   1:L PR[91] R[100]mm/sec CNT100;
   1:  PR[91,1] = PR[90,1] + 31.723;
   1:  PR[91,2] = PR[90,2] + -32.039;
   1:  PR[91,3] = PR[90,3] + 104.627;
   1:L PR[91] R[100]mm/sec CNT100;
   1:  PR[91,1] = PR[90,1] + 33.260;
   1:  PR[91,2] = PR[90,2] + -32.007;
   1:  PR[91,3] = PR[90,3] + 104.643;
   1:L PR[91] R[100]mm/sec CNT100;
   1:  PR[91,1] = PR[90,1] + 37.391;
   1:  PR[91,2] = PR[90,2] + -31.583;
   1:  PR[91,3] = PR[90,3] + 104.650;
   1:L PR[91] R[100]mm/sec CNT100;
   1:  PR[91,1] = PR[90,1] + 38.518;
   1:  PR[91,2] = PR[90,2] + -31.347;
   1:  PR[91,3] = PR[90,3] + 104.671;
   1:L PR[91] R[100]mm/sec CNT100;
   1:  PR[91,1] = PR[90,1] + 42.890;
   1:  PR[91,2] = PR[90,2] + -30.128;
   1:  PR[91,3] = PR[90,3] + 104.676;
   1:L PR[91] R[100]mm/sec CNT100;
   1:  PR[91,1] = PR[90,1] + 43.497;
   1:  PR[91,2] = PR[90,2] + -29.878;
   1:  PR[91,3] = PR[90,3] + 104.698;
   1:L PR[91] R[100]mm/sec CNT100;
   1:  PR[91,1] = PR[90,1] + 48.014;
   1:  PR[91,2] = PR[90,2] + -27.738;
   1:  PR[91,3] = PR[90,3] + 104.701;
   1:L PR[91] R[100]mm/sec CNT100;
   1:  PR[91,1] = PR[90,1] + 52.491;
   1:  PR[91,2] = PR[90,2] + -24.657;
   1:  PR[91,3] = PR[90,3] + 104.726;
   1:L PR[91] R[100]mm/sec CNT100;
   1:  PR[91,1] = PR[90,1] + 52.939;
   1:  PR[91,2] = PR[90,2] + -24.278;
   1:  PR[91,3] = PR[90,3] + 104.752;
   1:L PR[91] R[100]mm/sec CNT100;
   1:  PR[91,1] = PR[90,1] + 56.290;
   1:  PR[91,2] = PR[90,2] + -21.026;
   1:  PR[91,3] = PR[90,3] + 104.755;
   1:L PR[91] R[100]mm/sec CNT100;
   1:  PR[91,1] = PR[90,1] + 57.496;
   1:  PR[91,2] = PR[90,2] + -19.555;
   1:  PR[91,3] = PR[90,3] + 104.777;
   1:L PR[91] R[100]mm/sec CNT100;
   1:  PR[91,1] = PR[90,1] + 59.518;
   1:  PR[91,2] = PR[90,2] + -16.773;
   1:  PR[91,3] = PR[90,3] + 104.787;
   1:L PR[91] R[100]mm/sec CNT100;
   1:  PR[91,1] = PR[90,1] + 61.164;
   1:  PR[91,2] = PR[90,2] + -13.760;
   1:  PR[91,3] = PR[90,3] + 104.803;
   1:L PR[91] R[100]mm/sec CNT100;
   1:  PR[91,1] = PR[90,1] + 62.061;
   1:  PR[91,2] = PR[90,2] + -11.918;
   1:  PR[91,3] = PR[90,3] + 104.820;
   1:L PR[91] R[100]mm/sec CNT100;
   1:  PR[91,1] = PR[90,1] + 63.499;
   1:  PR[91,2] = PR[90,2] + -7.353;
   1:  PR[91,3] = PR[90,3] + 104.830;
   1:L PR[91] R[100]mm/sec CNT100;
   1:  PR[91,1] = PR[90,1] + 63.732;
   1:  PR[91,2] = PR[90,2] + -6.522;
   1:  PR[91,3] = PR[90,3] + 104.853;
   1:L PR[91] R[100]mm/sec CNT100;
   1:  PR[91,1] = PR[90,1] + 63.816;
   1:  PR[91,2] = PR[90,2] + -5.600;
   1:  PR[91,3] = PR[90,3] + 104.857;
   1:L PR[91] R[100]mm/sec CNT100;
   1:  PR[91,1] = PR[90,1] + 64.322;
   1:  PR[91,2] = PR[90,2] + -0.727;
   1:  PR[91,3] = PR[90,3] + 104.862;
   1:L PR[91] R[100]mm/sec CNT100;
   1:  PR[91,1] = PR[90,1] + 63.735;
   1:  PR[91,2] = PR[90,2] + 5.053;
   1:  PR[91,3] = PR[90,3] + 104.886;
   1:L PR[91] R[100]mm/sec CNT100;
   1:  PR[91,1] = PR[90,1] + 63.499;
   1:  PR[91,2] = PR[90,2] + 5.895;
   1:  PR[91,3] = PR[90,3] + 104.914;
   1:L PR[91] R[100]mm/sec CNT100;
   1:  PR[91,1] = PR[90,1] + 62.061;
   1:  PR[91,2] = PR[90,2] + 10.459;
   1:  PR[91,3] = PR[90,3] + 104.918;
   1:L PR[91] R[100]mm/sec CNT100;
   1:  PR[91,1] = PR[90,1] + 61.163;
   1:  PR[91,2] = PR[90,2] + 12.302;
   1:  PR[91,3] = PR[90,3] + 104.941;
   1:L PR[91] R[100]mm/sec CNT100;
   1:  PR[91,1] = PR[90,1] + 59.516;
   1:  PR[91,2] = PR[90,2] + 15.317;
   1:  PR[91,3] = PR[90,3] + 104.951;
   1:L PR[91] R[100]mm/sec CNT100;
   1:  PR[91,1] = PR[90,1] + 57.492;
   1:  PR[91,2] = PR[90,2] + 18.101;
   1:  PR[91,3] = PR[90,3] + 104.968;
   1:L PR[91] R[100]mm/sec CNT100;
   1:  PR[91,1] = PR[90,1] + 56.286;
   1:  PR[91,2] = PR[90,2] + 19.572;
   1:  PR[91,3] = PR[90,3] + 104.984;
   1:L PR[91] R[100]mm/sec CNT100;
   1:  PR[91,1] = PR[90,1] + 52.930;
   1:  PR[91,2] = PR[90,2] + 22.827;
   1:  PR[91,3] = PR[90,3] + 104.994;
   1:L PR[91] R[100]mm/sec CNT100;
   1:  PR[91,1] = PR[90,1] + 52.482;
   1:  PR[91,2] = PR[90,2] + 23.205;
   1:  PR[91,3] = PR[90,3] + 105.016;
   1:L PR[91] R[100]mm/sec CNT100;
   1:  PR[91,1] = PR[90,1] + 48.001;
   1:  PR[91,2] = PR[90,2] + 26.286;
   1:  PR[91,3] = PR[90,3] + 105.019;
   1:L PR[91] R[100]mm/sec CNT100;
   1:  PR[91,1] = PR[90,1] + 43.484;
   1:  PR[91,2] = PR[90,2] + 28.423;
   1:  PR[91,3] = PR[90,3] + 105.046;
   1:L PR[91] R[100]mm/sec CNT100;
   1:  PR[91,1] = PR[90,1] + 42.877;
   1:  PR[91,2] = PR[90,2] + 28.674;
   1:  PR[91,3] = PR[90,3] + 105.070;
   1:L PR[91] R[100]mm/sec CNT100;
   1:  PR[91,1] = PR[90,1] + 38.506;
   1:  PR[91,2] = PR[90,2] + 29.891;
   1:  PR[91,3] = PR[90,3] + 105.073;
   1:L PR[91] R[100]mm/sec CNT100;
   1:  PR[91,1] = PR[90,1] + 37.377;
   1:  PR[91,2] = PR[90,2] + 30.127;
   1:  PR[91,3] = PR[90,3] + 105.095;
   1:L PR[91] R[100]mm/sec CNT100;
   1:  PR[91,1] = PR[90,1] + 33.248;
   1:  PR[91,2] = PR[90,2] + 30.548;
   1:  PR[91,3] = PR[90,3] + 105.101;
   1:L PR[91] R[100]mm/sec CNT100;
   1:  PR[91,1] = PR[90,1] + 31.709;
   1:  PR[91,2] = PR[90,2] + 30.581;
   1:  PR[91,3] = PR[90,3] + 105.121;
   1:L PR[91] R[100]mm/sec CNT100;
   1:  PR[91,1] = PR[90,1] + 27.915;
   1:  PR[91,2] = PR[90,2] + 30.327;
   1:  PR[91,3] = PR[90,3] + 105.128;
   1:L PR[91] R[100]mm/sec CNT100;
   1:  PR[91,1] = PR[90,1] + 26.644;
   1:  PR[91,2] = PR[90,2] + 30.180;
   1:  PR[91,3] = PR[90,3] + 105.147;
   1:L PR[91] R[100]mm/sec CNT100;
   1:  PR[91,1] = PR[90,1] + 26.104;
   1:  PR[91,2] = PR[90,2] + 30.092;
   1:  PR[91,3] = PR[90,3] + 105.153;
   1:L PR[91] R[100]mm/sec CNT100;
   1:  PR[91,1] = PR[90,1] + 25.544;
   1:  PR[91,2] = PR[90,2] + 30.107;
   1:  PR[91,3] = PR[90,3] + 105.155;
   1:L PR[91] R[100]mm/sec CNT100;
   1:  PR[91,1] = PR[90,1] + 24.329;
   1:  PR[91,2] = PR[90,2] + 30.087;
   1:  PR[91,3] = PR[90,3] + 105.158;
   1:L PR[91] R[100]mm/sec CNT100;
   1:  PR[91,1] = PR[90,1] + 15.055;
   1:  PR[91,2] = PR[90,2] + 29.482;
   1:  PR[91,3] = PR[90,3] + 105.164;
   1:L PR[91] R[100]mm/sec CNT100;
   1:  PR[91,1] = PR[90,1] + 14.674;
   1:  PR[91,2] = PR[90,2] + 29.410;
   1:  PR[91,3] = PR[90,3] + 105.209;
   1:L PR[91] R[100]mm/sec CNT100;
   1:  PR[91,1] = PR[90,1] + 6.614;
   1:  PR[91,2] = PR[90,2] + 28.195;
   1:  PR[91,3] = PR[90,3] + 105.211;
   1:L PR[91] R[100]mm/sec CNT100;
   1:  PR[91,1] = PR[90,1] + 2.021;
   1:  PR[91,2] = PR[90,2] + 27.161;
   1:  PR[91,3] = PR[90,3] + 105.251;
   1:L PR[91] R[100]mm/sec CNT100;
   1:  PR[91,1] = PR[90,1] + -0.771;
   1:  PR[91,2] = PR[90,2] + 26.651;
   1:  PR[91,3] = PR[90,3] + 105.273;
   1:L PR[91] R[100]mm/sec CNT100;
   1:  PR[91,1] = PR[90,1] + -9.843;
   1:  PR[91,2] = PR[90,2] + 24.252;
   1:  PR[91,3] = PR[90,3] + 105.287;
   1:L PR[91] R[100]mm/sec CNT100;
   1:  PR[91,1] = PR[90,1] + -17.871;
   1:  PR[91,2] = PR[90,2] + 21.371;
   1:  PR[91,3] = PR[90,3] + 105.333;
   1:L PR[91] R[100]mm/sec CNT100;
   1:  PR[91,1] = PR[90,1] + -24.750;
   1:  PR[91,2] = PR[90,2] + 18.099;
   1:  PR[91,3] = PR[90,3] + 105.374;
   1:L PR[91] R[100]mm/sec CNT100;
   1:  PR[91,1] = PR[90,1] + -30.389;
   1:  PR[91,2] = PR[90,2] + 14.529;
   1:  PR[91,3] = PR[90,3] + 105.411;
   1:L PR[91] R[100]mm/sec CNT100;
   1:  PR[91,1] = PR[90,1] + -34.749;
   1:  PR[91,2] = PR[90,2] + 10.761;
   1:  PR[91,3] = PR[90,3] + 105.443;
   1:L PR[91] R[100]mm/sec CNT100;
   1:  PR[91,1] = PR[90,1] + -37.797;
   1:  PR[91,2] = PR[90,2] + 6.911;
   1:  PR[91,3] = PR[90,3] + 105.471;
   1:L PR[91] R[100]mm/sec CNT100;
   1:  PR[91] = PR[90];
   1:  PR[91,1] = PR[90,1] + -37.438;
   1:  PR[91,2] = PR[90,2] + 3.095;
   1:  PR[91,3] = PR[90,3] + 106.795;
   1:L PR[91] R[100]mm/sec CNT100;
   1:  PR[91,1] = PR[90,1] + -38.021;
   1:  PR[91,2] = PR[90,2] + -0.729;
   1:  PR[91,3] = PR[90,3] + 105.516;
   1:L PR[91] R[100]mm/sec CNT100;
   1:  PR[91,1] = PR[90,1] + -37.438;
   1:  PR[91,2] = PR[90,2] + -4.554;
   1:  PR[91,3] = PR[90,3] + 105.535;
   1:L PR[91] R[100]mm/sec CNT100;
   1:  PR[91,1] = PR[90,1] + -35.649;
   1:  PR[91,2] = PR[90,2] + -8.432;
   1:  PR[91,3] = PR[90,3] + 105.554;
   1:L PR[91] R[100]mm/sec CNT100;
   1:  PR[91,1] = PR[90,1] + -32.577;
   1:  PR[91,2] = PR[90,2] + -12.315;
   1:  PR[91,3] = PR[90,3] + 105.575;
   1:L PR[91] R[100]mm/sec CNT100;
   1:  PR[91,1] = PR[90,1] + -31.486;
   1:  PR[91,2] = PR[90,2] + -13.265;
   1:  PR[91,3] = PR[90,3] + 105.599;
   1:L PR[91] R[100]mm/sec CNT100;
   1:  PR[91,1] = PR[90,1] + -28.191;
   1:  PR[91,2] = PR[90,2] + -16.108;
   1:  PR[91,3] = PR[90,3] + 105.606;
   1:L PR[91] R[100]mm/sec CNT100;
   1:  PR[91,1] = PR[90,1] + -22.512;
   1:  PR[91,2] = PR[90,2] + -19.706;
   1:  PR[91,3] = PR[90,3] + 105.628;
   1:L PR[91] R[100]mm/sec CNT100;
   1:  PR[91,1] = PR[90,1] + -15.586;
   1:  PR[91,2] = PR[90,2] + -23.002;
   1:  PR[91,3] = PR[90,3] + 105.660;
   1:L PR[91] R[100]mm/sec CNT100;
   1:  PR[91,1] = PR[90,1] + -7.503;
   1:  PR[91,2] = PR[90,2] + -25.906;
   1:  PR[91,3] = PR[90,3] + 105.698;
   1:L PR[91] R[100]mm/sec CNT100;
   1:  PR[91,1] = PR[90,1] + 1.762;
   1:  PR[91,2] = PR[90,2] + -28.366;
   1:  PR[91,3] = PR[90,3] + 105.740;
   1:L PR[91] R[100]mm/sec CNT100;
   1:  PR[91,1] = PR[90,1] + 7.941;
   1:  PR[91,2] = PR[90,2] + -29.756;
   1:  PR[91,3] = PR[90,3] + 105.787;
   1:L PR[91] R[100]mm/sec CNT100;
   1:  PR[91,1] = PR[90,1] + 13.802;
   1:  PR[91,2] = PR[90,2] + -30.639;
   1:  PR[91,3] = PR[90,3] + 105.818;
   1:L PR[91] R[100]mm/sec CNT100;
   1:  PR[91,1] = PR[90,1] + 16.569;
   1:  PR[91,2] = PR[90,2] + -31.163;
   1:  PR[91,3] = PR[90,3] + 105.847;
   1:L PR[91] R[100]mm/sec CNT100;
   1:  PR[91,1] = PR[90,1] + 25.855;
   1:  PR[91,2] = PR[90,2] + -31.775;
   1:  PR[91,3] = PR[90,3] + 105.861;
   1:L PR[91] R[100]mm/sec CNT100;
   1:  PR[91,1] = PR[90,1] + 26.725;
   1:  PR[91,2] = PR[90,2] + -31.791;
   1:  PR[91,3] = PR[90,3] + 105.907;
   1:L PR[91] R[100]mm/sec CNT100;
   1:  PR[91,1] = PR[90,1] + 27.669;
   1:  PR[91,2] = PR[90,2] + -31.899;
   1:  PR[91,3] = PR[90,3] + 105.911;
   1:L PR[91] R[100]mm/sec CNT100;
   1:  PR[91,1] = PR[90,1] + 32.407;
   1:  PR[91,2] = PR[90,2] + -32.212;
   1:  PR[91,3] = PR[90,3] + 105.916;
   1:L PR[91] R[100]mm/sec CNT100;
   1:  PR[91,1] = PR[90,1] + 32.895;
   1:  PR[91,2] = PR[90,2] + -32.202;
   1:  PR[91,3] = PR[90,3] + 105.939;
   1:L PR[91] R[100]mm/sec CNT100;
   1:  PR[91,1] = PR[90,1] + 38.092;
   1:  PR[91,2] = PR[90,2] + -31.668;
   1:  PR[91,3] = PR[90,3] + 105.941;
   1:L PR[91] R[100]mm/sec CNT100;
   1:  PR[91,1] = PR[90,1] + 43.282;
   1:  PR[91,2] = PR[90,2] + -30.250;
   1:  PR[91,3] = PR[90,3] + 105.967;
   1:L PR[91] R[100]mm/sec CNT100;
   1:  PR[91,1] = PR[90,1] + 43.736;
   1:  PR[91,2] = PR[90,2] + -30.088;
   1:  PR[91,3] = PR[90,3] + 105.993;
   1:L PR[91] R[100]mm/sec CNT100;
   1:  PR[91,1] = PR[90,1] + 48.043;
   1:  PR[91,2] = PR[90,2] + -28.096;
   1:  PR[91,3] = PR[90,3] + 105.996;
   1:L PR[91] R[100]mm/sec CNT100;
   1:  PR[91,1] = PR[90,1] + 49.407;
   1:  PR[91,2] = PR[90,2] + -27.311;
   1:  PR[91,3] = PR[90,3] + 106.019;
   1:L PR[91] R[100]mm/sec CNT100;
   1:  PR[91,1] = PR[90,1] + 52.446;
   1:  PR[91,2] = PR[90,2] + -25.229;
   1:  PR[91,3] = PR[90,3] + 106.027;
   1:L PR[91] R[100]mm/sec CNT100;
   1:  PR[91,1] = PR[90,1] + 54.789;
   1:  PR[91,2] = PR[90,2] + -23.251;
   1:  PR[91,3] = PR[90,3] + 106.045;
   1:L PR[91] R[100]mm/sec CNT100;
   1:  PR[91,1] = PR[90,1] + 56.409;
   1:  PR[91,2] = PR[90,2] + -21.678;
   1:  PR[91,3] = PR[90,3] + 106.060;
   1:L PR[91] R[100]mm/sec CNT100;
   1:  PR[91,1] = PR[90,1] + 59.575;
   1:  PR[91,2] = PR[90,2] + -17.816;
   1:  PR[91,3] = PR[90,3] + 106.071;
   1:L PR[91] R[100]mm/sec CNT100;
   1:  PR[91,1] = PR[90,1] + 59.849;
   1:  PR[91,2] = PR[90,2] + -17.438;
   1:  PR[91,3] = PR[90,3] + 106.095;
   1:L PR[91] R[100]mm/sec CNT100;
   1:  PR[91,1] = PR[90,1] + 60.871;
   1:  PR[91,2] = PR[90,2] + -15.568;
   1:  PR[91,3] = PR[90,3] + 106.098;
   1:L PR[91] R[100]mm/sec CNT100;
   1:  PR[91,1] = PR[90,1] + 62.396;
   1:  PR[91,2] = PR[90,2] + -12.864;
   1:  PR[91,3] = PR[90,3] + 106.108;
   1:L PR[91] R[100]mm/sec CNT100;
   1:  PR[91,1] = PR[90,1] + 62.780;
   1:  PR[91,2] = PR[90,2] + -12.209;
   1:  PR[91,3] = PR[90,3] + 106.123;
   1:L PR[91] R[100]mm/sec CNT100;
   1:  PR[91,1] = PR[90,1] + 63.948;
   1:  PR[91,2] = PR[90,2] + -8.607;
   1:  PR[91,3] = PR[90,3] + 106.127;
   1:L PR[91] R[100]mm/sec CNT100;
   1:  PR[91,1] = PR[90,1] + 64.641;
   1:  PR[91,2] = PR[90,2] + -6.555;
   1:  PR[91,3] = PR[90,3] + 106.146;
   1:L PR[91] R[100]mm/sec CNT100;
   1:  PR[91,1] = PR[90,1] + 65.278;
   1:  PR[91,2] = PR[90,2] + -0.729;
   1:  PR[91,3] = PR[90,3] + 106.156;
   1:L PR[91] R[100]mm/sec CNT100;
   1:  PR[91,1] = PR[90,1] + 64.641;
   1:  PR[91,2] = PR[90,2] + 5.096;
   1:  PR[91,3] = PR[90,3] + 106.185;
   1:L PR[91] R[100]mm/sec CNT100;
   1:  PR[91,1] = PR[90,1] + 63.948;
   1:  PR[91,2] = PR[90,2] + 7.149;
   1:  PR[91,3] = PR[90,3] + 106.214;
   1:L PR[91] R[100]mm/sec CNT100;
   1:  PR[91,1] = PR[90,1] + 62.780;
   1:  PR[91,2] = PR[90,2] + 10.749;
   1:  PR[91,3] = PR[90,3] + 106.224;
   1:L PR[91] R[100]mm/sec CNT100;
   1:  PR[91,1] = PR[90,1] + 62.396;
   1:  PR[91,2] = PR[90,2] + 11.404;
   1:  PR[91,3] = PR[90,3] + 106.243;
   1:L PR[91] R[100]mm/sec CNT100;
   1:  PR[91,1] = PR[90,1] + 60.871;
   1:  PR[91,2] = PR[90,2] + 14.110;
   1:  PR[91,3] = PR[90,3] + 106.247;
   1:L PR[91] R[100]mm/sec CNT100;
   1:  PR[91,1] = PR[90,1] + 59.850;
   1:  PR[91,2] = PR[90,2] + 15.978;
   1:  PR[91,3] = PR[90,3] + 106.262;
   1:L PR[91] R[100]mm/sec CNT100;
   1:  PR[91,1] = PR[90,1] + 59.576;
   1:  PR[91,2] = PR[90,2] + 16.356;
   1:  PR[91,3] = PR[90,3] + 106.272;
   1:L PR[91] R[100]mm/sec CNT100;
   1:  PR[91,1] = PR[90,1] + 56.408;
   1:  PR[91,2] = PR[90,2] + 20.220;
   1:  PR[91,3] = PR[90,3] + 106.274;
   1:L PR[91] R[100]mm/sec CNT100;
   1:  PR[91,1] = PR[90,1] + 54.786;
   1:  PR[91,2] = PR[90,2] + 21.794;
   1:  PR[91,3] = PR[90,3] + 106.299;
   1:L PR[91] R[100]mm/sec CNT100;
   1:  PR[91,1] = PR[90,1] + 52.441;
   1:  PR[91,2] = PR[90,2] + 23.774;
   1:  PR[91,3] = PR[90,3] + 106.310;
   1:L PR[91] R[100]mm/sec CNT100;
   1:  PR[91,1] = PR[90,1] + 49.399;
   1:  PR[91,2] = PR[90,2] + 25.857;
   1:  PR[91,3] = PR[90,3] + 106.325;
   1:L PR[91] R[100]mm/sec CNT100;
   1:  PR[91,1] = PR[90,1] + 48.034;
   1:  PR[91,2] = PR[90,2] + 26.643;
   1:  PR[91,3] = PR[90,3] + 106.343;
   1:L PR[91] R[100]mm/sec CNT100;
   1:  PR[91,1] = PR[90,1] + 43.721;
   1:  PR[91,2] = PR[90,2] + 28.634;
   1:  PR[91,3] = PR[90,3] + 106.351;
   1:L PR[91] R[100]mm/sec CNT100;
   1:  PR[91,1] = PR[90,1] + 43.269;
   1:  PR[91,2] = PR[90,2] + 28.796;
   1:  PR[91,3] = PR[90,3] + 106.374;
   1:L PR[91] R[100]mm/sec CNT100;
   1:  PR[91,1] = PR[90,1] + 38.028;
   1:  PR[91,2] = PR[90,2] + 30.218;
   1:  PR[91,3] = PR[90,3] + 106.377;
   1:L PR[91] R[100]mm/sec CNT100;
   1:  PR[91,1] = PR[90,1] + 32.877;
   1:  PR[91,2] = PR[90,2] + 30.743;
   1:  PR[91,3] = PR[90,3] + 106.403;
   1:L PR[91] R[100]mm/sec CNT100;
   1:  PR[91,1] = PR[90,1] + 32.386;
   1:  PR[91,2] = PR[90,2] + 30.754;
   1:  PR[91,3] = PR[90,3] + 106.429;
   1:L PR[91] R[100]mm/sec CNT100;
   1:  PR[91,1] = PR[90,1] + 27.651;
   1:  PR[91,2] = PR[90,2] + 30.438;
   1:  PR[91,3] = PR[90,3] + 106.431;
   1:L PR[91] R[100]mm/sec CNT100;
   1:  PR[91,1] = PR[90,1] + 26.723;
   1:  PR[91,2] = PR[90,2] + 30.330;
   1:  PR[91,3] = PR[90,3] + 106.454;
   1:L PR[91] R[100]mm/sec CNT100;
   1:  PR[91,1] = PR[90,1] + 25.868;
   1:  PR[91,2] = PR[90,2] + 30.317;
   1:  PR[91,3] = PR[90,3] + 106.459;
   1:L PR[91] R[100]mm/sec CNT100;
   1:  PR[91,1] = PR[90,1] + 16.575;
   1:  PR[91,2] = PR[90,2] + 29.705;
   1:  PR[91,3] = PR[90,3] + 106.463;
   1:L PR[91] R[100]mm/sec CNT100;
   1:  PR[91,1] = PR[90,1] + 13.802;
   1:  PR[91,2] = PR[90,2] + 29.181;
   1:  PR[91,3] = PR[90,3] + 106.509;
   1:L PR[91] R[100]mm/sec CNT100;
   1:  PR[91,1] = PR[90,1] + 7.941;
   1:  PR[91,2] = PR[90,2] + 28.297;
   1:  PR[91,3] = PR[90,3] + 106.523;
   1:L PR[91] R[100]mm/sec CNT100;
   1:  PR[91,1] = PR[90,1] + 1.762;
   1:  PR[91,2] = PR[90,2] + 26.907;
   1:  PR[91,3] = PR[90,3] + 106.552;
   1:L PR[91] R[100]mm/sec CNT100;
   1:  PR[91,1] = PR[90,1] + -7.503;
   1:  PR[91,2] = PR[90,2] + 24.448;
   1:  PR[91,3] = PR[90,3] + 106.583;
   1:L PR[91] R[100]mm/sec CNT100;
   1:  PR[91,1] = PR[90,1] + -15.586;
   1:  PR[91,2] = PR[90,2] + 21.544;
   1:  PR[91,3] = PR[90,3] + 106.630;
   1:L PR[91] R[100]mm/sec CNT100;
   1:  PR[91,1] = PR[90,1] + -22.512;
   1:  PR[91,2] = PR[90,2] + 18.247;
   1:  PR[91,3] = PR[90,3] + 106.672;
   1:L PR[91] R[100]mm/sec CNT100;
   1:  PR[91,1] = PR[90,1] + -28.190;
   1:  PR[91,2] = PR[90,2] + 14.650;
   1:  PR[91,3] = PR[90,3] + 106.709;
   1:L PR[91] R[100]mm/sec CNT100;
   1:  PR[91,1] = PR[90,1] + -32.579;
   1:  PR[91,2] = PR[90,2] + 10.853;
   1:  PR[91,3] = PR[90,3] + 106.742;
   1:L PR[91] R[100]mm/sec CNT100;
   1:  PR[91,1] = PR[90,1] + -35.649;
   1:  PR[91,2] = PR[90,2] + 6.973;
   1:  PR[91,3] = PR[90,3] + 106.771;
   1:L PR[91] R[100]mm/sec CNT100;
   1:  PR[91] = PR[90];
   1:  PR[91,1] = PR[90,1] + -35.303;
   1:  PR[91,2] = PR[90,2] + 3.126;
   1:  PR[91,3] = PR[90,3] + 108.095;
   1:L PR[91] R[100]mm/sec CNT100;
   1:  PR[91,1] = PR[90,1] + -35.891;
   1:  PR[91,2] = PR[90,2] + -0.729;
   1:  PR[91,3] = PR[90,3] + 106.816;
   1:L PR[91] R[100]mm/sec CNT100;
   1:  PR[91,1] = PR[90,1] + -35.303;
   1:  PR[91,2] = PR[90,2] + -4.585;
   1:  PR[91,3] = PR[90,3] + 106.836;
   1:L PR[91] R[100]mm/sec CNT100;
   1:  PR[91,1] = PR[90,1] + -33.501;
   1:  PR[91,2] = PR[90,2] + -8.494;
   1:  PR[91,3] = PR[90,3] + 106.855;
   1:L PR[91] R[100]mm/sec CNT100;
   1:  PR[91,1] = PR[90,1] + -30.408;
   1:  PR[91,2] = PR[90,2] + -12.406;
   1:  PR[91,3] = PR[90,3] + 106.876;
   1:L PR[91] R[100]mm/sec CNT100;
   1:  PR[91,1] = PR[90,1] + -28.966;
   1:  PR[91,2] = PR[90,2] + -13.661;
   1:  PR[91,3] = PR[90,3] + 106.901;
   1:L PR[91] R[100]mm/sec CNT100;
   1:  PR[91,1] = PR[90,1] + -25.991;
   1:  PR[91,2] = PR[90,2] + -16.228;
   1:  PR[91,3] = PR[90,3] + 106.910;
   1:L PR[91] R[100]mm/sec CNT100;
   1:  PR[91,1] = PR[90,1] + -20.274;
   1:  PR[91,2] = PR[90,2] + -19.853;
   1:  PR[91,3] = PR[90,3] + 106.930;
   1:L PR[91] R[100]mm/sec CNT100;
   1:  PR[91,1] = PR[90,1] + -13.301;
   1:  PR[91,2] = PR[90,2] + -23.175;
   1:  PR[91,3] = PR[90,3] + 106.963;
   1:L PR[91] R[100]mm/sec CNT100;
   1:  PR[91,1] = PR[90,1] + -5.165;
   1:  PR[91,2] = PR[90,2] + -26.102;
   1:  PR[91,3] = PR[90,3] + 107.001;
   1:L PR[91] R[100]mm/sec CNT100;
   1:  PR[91,1] = PR[90,1] + 0.887;
   1:  PR[91,2] = PR[90,2] + -27.704;
   1:  PR[91,3] = PR[90,3] + 107.044;
   1:L PR[91] R[100]mm/sec CNT100;
   1:  PR[91,1] = PR[90,1] + 2.723;
   1:  PR[91,2] = PR[90,2] + -28.294;
   1:  PR[91,3] = PR[90,3] + 107.075;
   1:L PR[91] R[100]mm/sec CNT100;
   1:  PR[91,1] = PR[90,1] + 5.426;
   1:  PR[91,2] = PR[90,2] + -28.994;
   1:  PR[91,3] = PR[90,3] + 107.085;
   1:L PR[91] R[100]mm/sec CNT100;
   1:  PR[91,1] = PR[90,1] + 9.267;
   1:  PR[91,2] = PR[90,2] + -29.858;
   1:  PR[91,3] = PR[90,3] + 107.098;
   1:L PR[91] R[100]mm/sec CNT100;
   1:  PR[91,1] = PR[90,1] + 12.931;
   1:  PR[91,2] = PR[90,2] + -30.410;
   1:  PR[91,3] = PR[90,3] + 107.118;
   1:L PR[91] R[100]mm/sec CNT100;
   1:  PR[91,1] = PR[90,1] + 18.085;
   1:  PR[91,2] = PR[90,2] + -31.386;
   1:  PR[91,3] = PR[90,3] + 107.136;
   1:L PR[91] R[100]mm/sec CNT100;
   1:  PR[91,1] = PR[90,1] + 32.755;
   1:  PR[91,2] = PR[90,2] + -32.361;
   1:  PR[91,3] = PR[90,3] + 107.162;
   1:L PR[91] R[100]mm/sec CNT100;
   1:  PR[91,1] = PR[90,1] + 33.002;
   1:  PR[91,2] = PR[90,2] + -32.363;
   1:  PR[91,3] = PR[90,3] + 107.235;
   1:L PR[91] R[100]mm/sec CNT100;
   1:  PR[91,1] = PR[90,1] + 37.963;
   1:  PR[91,2] = PR[90,2] + -31.870;
   1:  PR[91,3] = PR[90,3] + 107.236;
   1:L PR[91] R[100]mm/sec CNT100;
   1:  PR[91,1] = PR[90,1] + 38.977;
   1:  PR[91,2] = PR[90,2] + -31.699;
   1:  PR[91,3] = PR[90,3] + 107.261;
   1:L PR[91] R[100]mm/sec CNT100;
   1:  PR[91,1] = PR[90,1] + 43.040;
   1:  PR[91,2] = PR[90,2] + -30.595;
   1:  PR[91,3] = PR[90,3] + 107.266;
   1:L PR[91] R[100]mm/sec CNT100;
   1:  PR[91,1] = PR[90,1] + 45.009;
   1:  PR[91,2] = PR[90,2] + -29.889;
   1:  PR[91,3] = PR[90,3] + 107.287;
   1:L PR[91] R[100]mm/sec CNT100;
   1:  PR[91,1] = PR[90,1] + 47.878;
   1:  PR[91,2] = PR[90,2] + -28.562;
   1:  PR[91,3] = PR[90,3] + 107.297;
   1:L PR[91] R[100]mm/sec CNT100;
   1:  PR[91,1] = PR[90,1] + 50.965;
   1:  PR[91,2] = PR[90,2] + -26.786;
   1:  PR[91,3] = PR[90,3] + 107.313;
   1:L PR[91] R[100]mm/sec CNT100;
   1:  PR[91,1] = PR[90,1] + 52.399;
   1:  PR[91,2] = PR[90,2] + -25.803;
   1:  PR[91,3] = PR[90,3] + 107.330;
   1:L PR[91] R[100]mm/sec CNT100;
   1:  PR[91,1] = PR[90,1] + 56.564;
   1:  PR[91,2] = PR[90,2] + -22.286;
   1:  PR[91,3] = PR[90,3] + 107.339;
   1:L PR[91] R[100]mm/sec CNT100;
   1:  PR[91,1] = PR[90,1] + 59.657;
   1:  PR[91,2] = PR[90,2] + -18.639;
   1:  PR[91,3] = PR[90,3] + 107.366;
   1:L PR[91] R[100]mm/sec CNT100;
   1:  PR[91,1] = PR[90,1] + 60.635;
   1:  PR[91,2] = PR[90,2] + -17.521;
   1:  PR[91,3] = PR[90,3] + 107.389;
   1:L PR[91] R[100]mm/sec CNT100;
   1:  PR[91,1] = PR[90,1] + 61.969;
   1:  PR[91,2] = PR[90,2] + -15.155;
   1:  PR[91,3] = PR[90,3] + 107.397;
   1:L PR[91] R[100]mm/sec CNT100;
   1:  PR[91,1] = PR[90,1] + 63.685;
   1:  PR[91,2] = PR[90,2] + -12.224;
   1:  PR[91,3] = PR[90,3] + 107.410;
   1:L PR[91] R[100]mm/sec CNT100;
   1:  PR[91,1] = PR[90,1] + 64.460;
   1:  PR[91,2] = PR[90,2] + -9.904;
   1:  PR[91,3] = PR[90,3] + 107.427;
   1:L PR[91] R[100]mm/sec CNT100;
   1:  PR[91,1] = PR[90,1] + 65.455;
   1:  PR[91,2] = PR[90,2] + -7.038;
   1:  PR[91,3] = PR[90,3] + 107.439;
   1:L PR[91] R[100]mm/sec CNT100;
   1:  PR[91,1] = PR[90,1] + 65.654;
   1:  PR[91,2] = PR[90,2] + -6.234;
   1:  PR[91,3] = PR[90,3] + 107.454;
   1:L PR[91] R[100]mm/sec CNT100;
   1:  PR[91,1] = PR[90,1] + 66.079;
   1:  PR[91,2] = PR[90,2] + -2.515;
   1:  PR[91,3] = PR[90,3] + 107.458;
   1:L PR[91] R[100]mm/sec CNT100;
   1:  PR[91,1] = PR[90,1] + 66.226;
   1:  PR[91,2] = PR[90,2] + -0.755;
   1:  PR[91,3] = PR[90,3] + 107.477;
   1:L PR[91] R[100]mm/sec CNT100;
   1:  PR[91,1] = PR[90,1] + 65.763;
   1:  PR[91,2] = PR[90,2] + 3.477;
   1:  PR[91,3] = PR[90,3] + 107.485;
   1:L PR[91] R[100]mm/sec CNT100;
   1:  PR[91,1] = PR[90,1] + 65.647;
   1:  PR[91,2] = PR[90,2] + 4.802;
   1:  PR[91,3] = PR[90,3] + 107.507;
   1:L PR[91] R[100]mm/sec CNT100;
   1:  PR[91,1] = PR[90,1] + 65.455;
   1:  PR[91,2] = PR[90,2] + 5.580;
   1:  PR[91,3] = PR[90,3] + 107.513;
   1:L PR[91] R[100]mm/sec CNT100;
   1:  PR[91,1] = PR[90,1] + 64.460;
   1:  PR[91,2] = PR[90,2] + 8.445;
   1:  PR[91,3] = PR[90,3] + 107.517;
   1:L PR[91] R[100]mm/sec CNT100;
   1:  PR[91,1] = PR[90,1] + 63.684;
   1:  PR[91,2] = PR[90,2] + 10.767;
   1:  PR[91,3] = PR[90,3] + 107.532;
   1:L PR[91] R[100]mm/sec CNT100;
   1:  PR[91,1] = PR[90,1] + 61.969;
   1:  PR[91,2] = PR[90,2] + 13.697;
   1:  PR[91,3] = PR[90,3] + 107.544;
   1:L PR[91] R[100]mm/sec CNT100;
   1:  PR[91,1] = PR[90,1] + 60.635;
   1:  PR[91,2] = PR[90,2] + 16.062;
   1:  PR[91,3] = PR[90,3] + 107.561;
   1:L PR[91] R[100]mm/sec CNT100;
   1:  PR[91,1] = PR[90,1] + 59.657;
   1:  PR[91,2] = PR[90,2] + 17.180;
   1:  PR[91,3] = PR[90,3] + 107.574;
   1:L PR[91] R[100]mm/sec CNT100;
   1:  PR[91,1] = PR[90,1] + 56.587;
   1:  PR[91,2] = PR[90,2] + 20.805;
   1:  PR[91,3] = PR[90,3] + 107.582;
   1:L PR[91] R[100]mm/sec CNT100;
   1:  PR[91,1] = PR[90,1] + 52.398;
   1:  PR[91,2] = PR[90,2] + 24.345;
   1:  PR[91,3] = PR[90,3] + 107.605;
   1:L PR[91] R[100]mm/sec CNT100;
   1:  PR[91,1] = PR[90,1] + 50.963;
   1:  PR[91,2] = PR[90,2] + 25.328;
   1:  PR[91,3] = PR[90,3] + 107.632;
   1:L PR[91] R[100]mm/sec CNT100;
   1:  PR[91,1] = PR[90,1] + 47.874;
   1:  PR[91,2] = PR[90,2] + 27.106;
   1:  PR[91,3] = PR[90,3] + 107.641;
   1:L PR[91] R[100]mm/sec CNT100;
   1:  PR[91,1] = PR[90,1] + 45.001;
   1:  PR[91,2] = PR[90,2] + 28.433;
   1:  PR[91,3] = PR[90,3] + 107.659;
   1:L PR[91] R[100]mm/sec CNT100;
   1:  PR[91,1] = PR[90,1] + 43.031;
   1:  PR[91,2] = PR[90,2] + 29.139;
   1:  PR[91,3] = PR[90,3] + 107.674;
   1:L PR[91] R[100]mm/sec CNT100;
   1:  PR[91,1] = PR[90,1] + 38.962;
   1:  PR[91,2] = PR[90,2] + 30.243;
   1:  PR[91,3] = PR[90,3] + 107.685;
   1:L PR[91] R[100]mm/sec CNT100;
   1:  PR[91,1] = PR[90,1] + 37.948;
   1:  PR[91,2] = PR[90,2] + 30.414;
   1:  PR[91,3] = PR[90,3] + 107.705;
   1:L PR[91] R[100]mm/sec CNT100;
   1:  PR[91,1] = PR[90,1] + 32.980;
   1:  PR[91,2] = PR[90,2] + 30.905;
   1:  PR[91,3] = PR[90,3] + 107.710;
   1:L PR[91] R[100]mm/sec CNT100;
   1:  PR[91,1] = PR[90,1] + 32.734;
   1:  PR[91,2] = PR[90,2] + 30.903;
   1:  PR[91,3] = PR[90,3] + 107.735;
   1:L PR[91] R[100]mm/sec CNT100;
   1:  PR[91,1] = PR[90,1] + 18.096;
   1:  PR[91,2] = PR[90,2] + 29.928;
   1:  PR[91,3] = PR[90,3] + 107.736;
   1:L PR[91] R[100]mm/sec CNT100;
   1:  PR[91,1] = PR[90,1] + 12.931;
   1:  PR[91,2] = PR[90,2] + 28.952;
   1:  PR[91,3] = PR[90,3] + 107.809;
   1:L PR[91] R[100]mm/sec CNT100;
   1:  PR[91,1] = PR[90,1] + 9.268;
   1:  PR[91,2] = PR[90,2] + 28.399;
   1:  PR[91,3] = PR[90,3] + 107.835;
   1:L PR[91] R[100]mm/sec CNT100;
   1:  PR[91,1] = PR[90,1] + 5.427;
   1:  PR[91,2] = PR[90,2] + 27.535;
   1:  PR[91,3] = PR[90,3] + 107.853;
   1:L PR[91] R[100]mm/sec CNT100;
   1:  PR[91,1] = PR[90,1] + 2.723;
   1:  PR[91,2] = PR[90,2] + 26.836;
   1:  PR[91,3] = PR[90,3] + 107.873;
   1:L PR[91] R[100]mm/sec CNT100;
   1:  PR[91,1] = PR[90,1] + 0.887;
   1:  PR[91,2] = PR[90,2] + 26.246;
   1:  PR[91,3] = PR[90,3] + 107.887;
   1:L PR[91] R[100]mm/sec CNT100;
   1:  PR[91,1] = PR[90,1] + -5.165;
   1:  PR[91,2] = PR[90,2] + 24.643;
   1:  PR[91,3] = PR[90,3] + 107.896;
   1:L PR[91] R[100]mm/sec CNT100;
   1:  PR[91,1] = PR[90,1] + -13.301;
   1:  PR[91,2] = PR[90,2] + 21.717;
   1:  PR[91,3] = PR[90,3] + 107.927;
   1:L PR[91] R[100]mm/sec CNT100;
   1:  PR[91,1] = PR[90,1] + -20.276;
   1:  PR[91,2] = PR[90,2] + 18.394;
   1:  PR[91,3] = PR[90,3] + 107.970;
   1:L PR[91] R[100]mm/sec CNT100;
   1:  PR[91,1] = PR[90,1] + -23.310;
   1:  PR[91,2] = PR[90,2] + 16.479;
   1:  PR[91,3] = PR[90,3] + 108.008;
   1:L PR[91] R[100]mm/sec CNT100;
   1:  PR[91,1] = PR[90,1] + -25.988;
   1:  PR[91,2] = PR[90,2] + 14.772;
   1:  PR[91,3] = PR[90,3] + 108.026;
   1:L PR[91] R[100]mm/sec CNT100;
   1:  PR[91,1] = PR[90,1] + -30.410;
   1:  PR[91,2] = PR[90,2] + 10.945;
   1:  PR[91,3] = PR[90,3] + 108.041;
   1:L PR[91] R[100]mm/sec CNT100;
   1:  PR[91,1] = PR[90,1] + -33.501;
   1:  PR[91,2] = PR[90,2] + 7.035;
   1:  PR[91,3] = PR[90,3] + 108.070;
   1:L PR[91] R[100]mm/sec CNT100;
   1:  PR[91] = PR[90];
   1:  PR[91,1] = PR[90,1] + -33.168;
   1:  PR[91,2] = PR[90,2] + 3.157;
   1:  PR[91,3] = PR[90,3] + 109.395;
   1:L PR[91] R[100]mm/sec CNT100;
   1:  PR[91,1] = PR[90,1] + -33.760;
   1:  PR[91,2] = PR[90,2] + -0.729;
   1:  PR[91,3] = PR[90,3] + 108.117;
   1:L PR[91] R[100]mm/sec CNT100;
   1:  PR[91,1] = PR[90,1] + -33.168;
   1:  PR[91,2] = PR[90,2] + -4.616;
   1:  PR[91,3] = PR[90,3] + 108.136;
   1:L PR[91] R[100]mm/sec CNT100;
   1:  PR[91,1] = PR[90,1] + -31.353;
   1:  PR[91,2] = PR[90,2] + -8.556;
   1:  PR[91,3] = PR[90,3] + 108.156;
   1:L PR[91] R[100]mm/sec CNT100;
   1:  PR[91,1] = PR[90,1] + -28.238;
   1:  PR[91,2] = PR[90,2] + -12.497;
   1:  PR[91,3] = PR[90,3] + 108.177;
   1:L PR[91] R[100]mm/sec CNT100;
   1:  PR[91,1] = PR[90,1] + -26.447;
   1:  PR[91,2] = PR[90,2] + -14.057;
   1:  PR[91,3] = PR[90,3] + 108.203;
   1:L PR[91] R[100]mm/sec CNT100;
   1:  PR[91,1] = PR[90,1] + -23.792;
   1:  PR[91,2] = PR[90,2] + -16.348;
   1:  PR[91,3] = PR[90,3] + 108.214;
   1:L PR[91] R[100]mm/sec CNT100;
   1:  PR[91,1] = PR[90,1] + -18.036;
   1:  PR[91,2] = PR[90,2] + -20.001;
   1:  PR[91,3] = PR[90,3] + 108.232;
   1:L PR[91] R[100]mm/sec CNT100;
   1:  PR[91,1] = PR[90,1] + -11.016;
   1:  PR[91,2] = PR[90,2] + -23.349;
   1:  PR[91,3] = PR[90,3] + 108.266;
   1:L PR[91] R[100]mm/sec CNT100;
   1:  PR[91,1] = PR[90,1] + -2.826;
   1:  PR[91,2] = PR[90,2] + -26.298;
   1:  PR[91,3] = PR[90,3] + 108.305;
   1:L PR[91] R[100]mm/sec CNT100;
   1:  PR[91,1] = PR[90,1] + 0.239;
   1:  PR[91,2] = PR[90,2] + -27.109;
   1:  PR[91,3] = PR[90,3] + 108.348;
   1:L PR[91] R[100]mm/sec CNT100;
   1:  PR[91,1] = PR[90,1] + 3.791;
   1:  PR[91,2] = PR[90,2] + -28.251;
   1:  PR[91,3] = PR[90,3] + 108.364;
   1:L PR[91] R[100]mm/sec CNT100;
   1:  PR[91,1] = PR[90,1] + 9.096;
   1:  PR[91,2] = PR[90,2] + -29.623;
   1:  PR[91,3] = PR[90,3] + 108.383;
   1:L PR[91] R[100]mm/sec CNT100;
   1:  PR[91,1] = PR[90,1] + 10.594;
   1:  PR[91,2] = PR[90,2] + -29.960;
   1:  PR[91,3] = PR[90,3] + 108.410;
   1:L PR[91] R[100]mm/sec CNT100;
   1:  PR[91,1] = PR[90,1] + 12.059;
   1:  PR[91,2] = PR[90,2] + -30.181;
   1:  PR[91,3] = PR[90,3] + 108.417;
   1:L PR[91] R[100]mm/sec CNT100;
   1:  PR[91,1] = PR[90,1] + 19.601;
   1:  PR[91,2] = PR[90,2] + -31.608;
   1:  PR[91,3] = PR[90,3] + 108.425;
   1:L PR[91] R[100]mm/sec CNT100;
   1:  PR[91,1] = PR[90,1] + 32.469;
   1:  PR[91,2] = PR[90,2] + -32.466;
   1:  PR[91,3] = PR[90,3] + 108.463;
   1:L PR[91] R[100]mm/sec CNT100;
   1:  PR[91,1] = PR[90,1] + 33.818;
   1:  PR[91,2] = PR[90,2] + -32.475;
   1:  PR[91,3] = PR[90,3] + 108.527;
   1:L PR[91] R[100]mm/sec CNT100;
   1:  PR[91,1] = PR[90,1] + 37.673;
   1:  PR[91,2] = PR[90,2] + -32.092;
   1:  PR[91,3] = PR[90,3] + 108.534;
   1:L PR[91] R[100]mm/sec CNT100;
   1:  PR[91,1] = PR[90,1] + 40.001;
   1:  PR[91,2] = PR[90,2] + -31.699;
   1:  PR[91,3] = PR[90,3] + 108.554;
   1:L PR[91] R[100]mm/sec CNT100;
   1:  PR[91,1] = PR[90,1] + 42.797;
   1:  PR[91,2] = PR[90,2] + -30.939;
   1:  PR[91,3] = PR[90,3] + 108.565;
   1:L PR[91] R[100]mm/sec CNT100;
   1:  PR[91,1] = PR[90,1] + 46.282;
   1:  PR[91,2] = PR[90,2] + -29.690;
   1:  PR[91,3] = PR[90,3] + 108.580;
   1:L PR[91] R[100]mm/sec CNT100;
   1:  PR[91,1] = PR[90,1] + 47.714;
   1:  PR[91,2] = PR[90,2] + -29.028;
   1:  PR[91,3] = PR[90,3] + 108.598;
   1:L PR[91] R[100]mm/sec CNT100;
   1:  PR[91,1] = PR[90,1] + 52.439;
   1:  PR[91,2] = PR[90,2] + -26.310;
   1:  PR[91,3] = PR[90,3] + 108.606;
   1:L PR[91] R[100]mm/sec CNT100;
   1:  PR[91,1] = PR[90,1] + 56.151;
   1:  PR[91,2] = PR[90,2] + -23.284;
   1:  PR[91,3] = PR[90,3] + 108.633;
   1:L PR[91] R[100]mm/sec CNT100;
   1:  PR[91,1] = PR[90,1] + 57.391;
   1:  PR[91,2] = PR[90,2] + -22.295;
   1:  PR[91,3] = PR[90,3] + 108.657;
   1:L PR[91] R[100]mm/sec CNT100;
   1:  PR[91,1] = PR[90,1] + 59.089;
   1:  PR[91,2] = PR[90,2] + -20.291;
   1:  PR[91,3] = PR[90,3] + 108.665;
   1:L PR[91] R[100]mm/sec CNT100;
   1:  PR[91,1] = PR[90,1] + 61.490;
   1:  PR[91,2] = PR[90,2] + -17.544;
   1:  PR[91,3] = PR[90,3] + 108.678;
   1:L PR[91] R[100]mm/sec CNT100;
   1:  PR[91,1] = PR[90,1] + 63.751;
   1:  PR[91,2] = PR[90,2] + -13.654;
   1:  PR[91,3] = PR[90,3] + 108.696;
   1:L PR[91] R[100]mm/sec CNT100;
   1:  PR[91,1] = PR[90,1] + 64.329;
   1:  PR[91,2] = PR[90,2] + -12.776;
   1:  PR[91,3] = PR[90,3] + 108.719;
   1:L PR[91] R[100]mm/sec CNT100;
   1:  PR[91,1] = PR[90,1] + 65.406;
   1:  PR[91,2] = PR[90,2] + -10.217;
   1:  PR[91,3] = PR[90,3] + 108.724;
   1:L PR[91] R[100]mm/sec CNT100;
   1:  PR[91,1] = PR[90,1] + 65.848;
   1:  PR[91,2] = PR[90,2] + -8.943;
   1:  PR[91,3] = PR[90,3] + 108.738;
   1:L PR[91] R[100]mm/sec CNT100;
   1:  PR[91,1] = PR[90,1] + 66.790;
   1:  PR[91,2] = PR[90,2] + -5.141;
   1:  PR[91,3] = PR[90,3] + 108.745;
   1:L PR[91] R[100]mm/sec CNT100;
   1:  PR[91,1] = PR[90,1] + 67.153;
   1:  PR[91,2] = PR[90,2] + -0.729;
   1:  PR[91,3] = PR[90,3] + 108.764;
   1:L PR[91] R[100]mm/sec CNT100;
   1:  PR[91,1] = PR[90,1] + 66.790;
   1:  PR[91,2] = PR[90,2] + 3.683;
   1:  PR[91,3] = PR[90,3] + 108.786;
   1:L PR[91] R[100]mm/sec CNT100;
   1:  PR[91,1] = PR[90,1] + 65.848;
   1:  PR[91,2] = PR[90,2] + 7.484;
   1:  PR[91,3] = PR[90,3] + 108.808;
   1:L PR[91] R[100]mm/sec CNT100;
   1:  PR[91,1] = PR[90,1] + 65.406;
   1:  PR[91,2] = PR[90,2] + 8.758;
   1:  PR[91,3] = PR[90,3] + 108.828;
   1:L PR[91] R[100]mm/sec CNT100;
   1:  PR[91,1] = PR[90,1] + 64.312;
   1:  PR[91,2] = PR[90,2] + 11.357;
   1:  PR[91,3] = PR[90,3] + 108.835;
   1:L PR[91] R[100]mm/sec CNT100;
   1:  PR[91,1] = PR[90,1] + 61.839;
   1:  PR[91,2] = PR[90,2] + 15.481;
   1:  PR[91,3] = PR[90,3] + 108.849;
   1:L PR[91] R[100]mm/sec CNT100;
   1:  PR[91,1] = PR[90,1] + 61.487;
   1:  PR[91,2] = PR[90,2] + 16.090;
   1:  PR[91,3] = PR[90,3] + 108.873;
   1:L PR[91] R[100]mm/sec CNT100;
   1:  PR[91,1] = PR[90,1] + 59.088;
   1:  PR[91,2] = PR[90,2] + 18.833;
   1:  PR[91,3] = PR[90,3] + 108.876;
   1:L PR[91] R[100]mm/sec CNT100;
   1:  PR[91,1] = PR[90,1] + 57.391;
   1:  PR[91,2] = PR[90,2] + 20.836;
   1:  PR[91,3] = PR[90,3] + 108.894;
   1:L PR[91] R[100]mm/sec CNT100;
   1:  PR[91,1] = PR[90,1] + 56.151;
   1:  PR[91,2] = PR[90,2] + 21.824;
   1:  PR[91,3] = PR[90,3] + 108.907;
   1:L PR[91] R[100]mm/sec CNT100;
   1:  PR[91,1] = PR[90,1] + 52.443;
   1:  PR[91,2] = PR[90,2] + 24.849;
   1:  PR[91,3] = PR[90,3] + 108.915;
   1:L PR[91] R[100]mm/sec CNT100;
   1:  PR[91,1] = PR[90,1] + 47.714;
   1:  PR[91,2] = PR[90,2] + 27.570;
   1:  PR[91,3] = PR[90,3] + 108.939;
   1:L PR[91] R[100]mm/sec CNT100;
   1:  PR[91,1] = PR[90,1] + 46.280;
   1:  PR[91,2] = PR[90,2] + 28.232;
   1:  PR[91,3] = PR[90,3] + 108.966;
   1:L PR[91] R[100]mm/sec CNT100;
   1:  PR[91,1] = PR[90,1] + 42.792;
   1:  PR[91,2] = PR[90,2] + 29.483;
   1:  PR[91,3] = PR[90,3] + 108.974;
   1:L PR[91] R[100]mm/sec CNT100;
   1:  PR[91,1] = PR[90,1] + 39.992;
   1:  PR[91,2] = PR[90,2] + 30.242;
   1:  PR[91,3] = PR[90,3] + 108.993;
   1:L PR[91] R[100]mm/sec CNT100;
   1:  PR[91,1] = PR[90,1] + 37.663;
   1:  PR[91,2] = PR[90,2] + 30.635;
   1:  PR[91,3] = PR[90,3] + 109.007;
   1:L PR[91] R[100]mm/sec CNT100;
   1:  PR[91,1] = PR[90,1] + 33.803;
   1:  PR[91,2] = PR[90,2] + 31.016;
   1:  PR[91,3] = PR[90,3] + 109.019;
   1:L PR[91] R[100]mm/sec CNT100;
   1:  PR[91,1] = PR[90,1] + 32.449;
   1:  PR[91,2] = PR[90,2] + 31.007;
   1:  PR[91,3] = PR[90,3] + 109.038;
   1:L PR[91] R[100]mm/sec CNT100;
   1:  PR[91,1] = PR[90,1] + 19.615;
   1:  PR[91,2] = PR[90,2] + 30.152;
   1:  PR[91,3] = PR[90,3] + 109.045;
   1:L PR[91] R[100]mm/sec CNT100;
   1:  PR[91,1] = PR[90,1] + 12.059;
   1:  PR[91,2] = PR[90,2] + 28.723;
   1:  PR[91,3] = PR[90,3] + 109.109;
   1:L PR[91] R[100]mm/sec CNT100;
   1:  PR[91,1] = PR[90,1] + 10.594;
   1:  PR[91,2] = PR[90,2] + 28.502;
   1:  PR[91,3] = PR[90,3] + 109.148;
   1:L PR[91] R[100]mm/sec CNT100;
   1:  PR[91,1] = PR[90,1] + 9.097;
   1:  PR[91,2] = PR[90,2] + 28.165;
   1:  PR[91,3] = PR[90,3] + 109.155;
   1:L PR[91] R[100]mm/sec CNT100;
   1:  PR[91,1] = PR[90,1] + 3.791;
   1:  PR[91,2] = PR[90,2] + 26.792;
   1:  PR[91,3] = PR[90,3] + 109.163;
   1:L PR[91] R[100]mm/sec CNT100;
   1:  PR[91,1] = PR[90,1] + 0.239;
   1:  PR[91,2] = PR[90,2] + 25.650;
   1:  PR[91,3] = PR[90,3] + 109.190;
   1:L PR[91] R[100]mm/sec CNT100;
   1:  PR[91,1] = PR[90,1] + -2.826;
   1:  PR[91,2] = PR[90,2] + 24.839;
   1:  PR[91,3] = PR[90,3] + 109.209;
   1:L PR[91] R[100]mm/sec CNT100;
   1:  PR[91,1] = PR[90,1] + -11.016;
   1:  PR[91,2] = PR[90,2] + 21.890;
   1:  PR[91,3] = PR[90,3] + 109.224;
   1:L PR[91] R[100]mm/sec CNT100;
   1:  PR[91,1] = PR[90,1] + -18.038;
   1:  PR[91,2] = PR[90,2] + 18.541;
   1:  PR[91,3] = PR[90,3] + 109.268;
   1:L PR[91] R[100]mm/sec CNT100;
   1:  PR[91,1] = PR[90,1] + -20.653;
   1:  PR[91,2] = PR[90,2] + 16.891;
   1:  PR[91,3] = PR[90,3] + 109.307;
   1:L PR[91] R[100]mm/sec CNT100;
   1:  PR[91,1] = PR[90,1] + -23.788;
   1:  PR[91,2] = PR[90,2] + 14.892;
   1:  PR[91,3] = PR[90,3] + 109.322;
   1:L PR[91] R[100]mm/sec CNT100;
   1:  PR[91,1] = PR[90,1] + -28.240;
   1:  PR[91,2] = PR[90,2] + 11.036;
   1:  PR[91,3] = PR[90,3] + 109.341;
   1:L PR[91] R[100]mm/sec CNT100;
   1:  PR[91,1] = PR[90,1] + -31.353;
   1:  PR[91,2] = PR[90,2] + 7.097;
   1:  PR[91,3] = PR[90,3] + 109.370;
   1:L PR[91] R[100]mm/sec CNT100;
   1:  PR[91] = PR[90];
   1:  PR[91,1] = PR[90,1] + -31.033;
   1:  PR[91,2] = PR[90,2] + 3.188;
   1:  PR[91,3] = PR[90,3] + 110.695;
   1:L PR[91] R[100]mm/sec CNT100;
   1:  PR[91,1] = PR[90,1] + -31.630;
   1:  PR[91,2] = PR[90,2] + -0.729;
   1:  PR[91,3] = PR[90,3] + 109.417;
   1:L PR[91] R[100]mm/sec CNT100;
   1:  PR[91,1] = PR[90,1] + -31.033;
   1:  PR[91,2] = PR[90,2] + -4.647;
   1:  PR[91,3] = PR[90,3] + 109.437;
   1:L PR[91] R[100]mm/sec CNT100;
   1:  PR[91,1] = PR[90,1] + -29.205;
   1:  PR[91,2] = PR[90,2] + -8.618;
   1:  PR[91,3] = PR[90,3] + 109.457;
   1:L PR[91] R[100]mm/sec CNT100;
   1:  PR[91,1] = PR[90,1] + -26.069;
   1:  PR[91,2] = PR[90,2] + -12.589;
   1:  PR[91,3] = PR[90,3] + 109.479;
   1:L PR[91] R[100]mm/sec CNT100;
   1:  PR[91,1] = PR[90,1] + -23.927;
   1:  PR[91,2] = PR[90,2] + -14.454;
   1:  PR[91,3] = PR[90,3] + 109.504;
   1:L PR[91] R[100]mm/sec CNT100;
   1:  PR[91,1] = PR[90,1] + -21.592;
   1:  PR[91,2] = PR[90,2] + -16.469;
   1:  PR[91,3] = PR[90,3] + 109.519;
   1:L PR[91] R[100]mm/sec CNT100;
   1:  PR[91,1] = PR[90,1] + -15.798;
   1:  PR[91,2] = PR[90,2] + -20.149;
   1:  PR[91,3] = PR[90,3] + 109.534;
   1:L PR[91] R[100]mm/sec CNT100;
   1:  PR[91,1] = PR[90,1] + -8.731;
   1:  PR[91,2] = PR[90,2] + -23.521;
   1:  PR[91,3] = PR[90,3] + 109.569;
   1:L PR[91] R[100]mm/sec CNT100;
   1:  PR[91,1] = PR[90,1] + -0.438;
   1:  PR[91,2] = PR[90,2] + -26.511;
   1:  PR[91,3] = PR[90,3] + 109.608;
   1:L PR[91] R[100]mm/sec CNT100;
   1:  PR[91,1] = PR[90,1] + 4.858;
   1:  PR[91,2] = PR[90,2] + -28.207;
   1:  PR[91,3] = PR[90,3] + 109.652;
   1:L PR[91] R[100]mm/sec CNT100;
   1:  PR[91,1] = PR[90,1] + 11.413;
   1:  PR[91,2] = PR[90,2] + -29.903;
   1:  PR[91,3] = PR[90,3] + 109.680;
   1:L PR[91] R[100]mm/sec CNT100;
   1:  PR[91,1] = PR[90,1] + 12.090;
   1:  PR[91,2] = PR[90,2] + -30.123;
   1:  PR[91,3] = PR[90,3] + 109.714;
   1:L PR[91] R[100]mm/sec CNT100;
   1:  PR[91,1] = PR[90,1] + 21.116;
   1:  PR[91,2] = PR[90,2] + -31.831;
   1:  PR[91,3] = PR[90,3] + 109.718;
   1:L PR[91] R[100]mm/sec CNT100;
   1:  PR[91,1] = PR[90,1] + 32.183;
   1:  PR[91,2] = PR[90,2] + -32.570;
   1:  PR[91,3] = PR[90,3] + 109.764;
   1:L PR[91] R[100]mm/sec CNT100;
   1:  PR[91,1] = PR[90,1] + 34.634;
   1:  PR[91,2] = PR[90,2] + -32.587;
   1:  PR[91,3] = PR[90,3] + 109.820;
   1:L PR[91] R[100]mm/sec CNT100;
   1:  PR[91,1] = PR[90,1] + 37.384;
   1:  PR[91,2] = PR[90,2] + -32.313;
   1:  PR[91,3] = PR[90,3] + 109.832;
   1:L PR[91] R[100]mm/sec CNT100;
   1:  PR[91,1] = PR[90,1] + 41.025;
   1:  PR[91,2] = PR[90,2] + -31.699;
   1:  PR[91,3] = PR[90,3] + 109.846;
   1:L PR[91] R[100]mm/sec CNT100;
   1:  PR[91,1] = PR[90,1] + 42.554;
   1:  PR[91,2] = PR[90,2] + -31.284;
   1:  PR[91,3] = PR[90,3] + 109.865;
   1:L PR[91] R[100]mm/sec CNT100;
   1:  PR[91,1] = PR[90,1] + 47.555;
   1:  PR[91,2] = PR[90,2] + -29.492;
   1:  PR[91,3] = PR[90,3] + 109.873;
   1:L PR[91] R[100]mm/sec CNT100;
   1:  PR[91,1] = PR[90,1] + 47.563;
   1:  PR[91,2] = PR[90,2] + -29.488;
   1:  PR[91,3] = PR[90,3] + 109.900;
   1:L PR[91] R[100]mm/sec CNT100;
   1:  PR[91,1] = PR[90,1] + 53.203;
   1:  PR[91,2] = PR[90,2] + -26.355;
   1:L PR[91] R[100]mm/sec CNT100;
   1:  PR[91,1] = PR[90,1] + 55.545;
   1:  PR[91,2] = PR[90,2] + -24.445;
   1:  PR[91,3] = PR[90,3] + 109.932;
   1:L PR[91] R[100]mm/sec CNT100;
   1:  PR[91,1] = PR[90,1] + 58.193;
   1:  PR[91,2] = PR[90,2] + -22.332;
   1:  PR[91,3] = PR[90,3] + 109.947;
   1:L PR[91] R[100]mm/sec CNT100;
   1:  PR[91,1] = PR[90,1] + 59.270;
   1:  PR[91,2] = PR[90,2] + -21.086;
   1:  PR[91,3] = PR[90,3] + 109.964;
   1:L PR[91] R[100]mm/sec CNT100;
   1:  PR[91,1] = PR[90,1] + 61.513;
   1:  PR[91,2] = PR[90,2] + -18.578;
   1:  PR[91,3] = PR[90,3] + 109.973;
   1:L PR[91] R[100]mm/sec CNT100;
   1:  PR[91,1] = PR[90,1] + 62.353;
   1:  PR[91,2] = PR[90,2] + -17.590;
   1:  PR[91,3] = PR[90,3] + 109.989;
   1:L PR[91] R[100]mm/sec CNT100;
   1:  PR[91,1] = PR[90,1] + 63.404;
   1:  PR[91,2] = PR[90,2] + -15.783;
   1:  PR[91,3] = PR[90,3] + 109.996;
   1:L PR[91] R[100]mm/sec CNT100;
   1:  PR[91,1] = PR[90,1] + 64.827;
   1:  PR[91,2] = PR[90,2] + -13.617;
   1:  PR[91,3] = PR[90,3] + 110.007;
   1:L PR[91] R[100]mm/sec CNT100;
   1:  PR[91,1] = PR[90,1] + 66.603;
   1:  PR[91,2] = PR[90,2] + -9.430;
   1:  PR[91,3] = PR[90,3] + 110.020;
   1:L PR[91] R[100]mm/sec CNT100;
   1:  PR[91,1] = PR[90,1] + 67.642;
   1:  PR[91,2] = PR[90,2] + -5.250;
   1:  PR[91,3] = PR[90,3] + 110.042;
   1:L PR[91] R[100]mm/sec CNT100;
   1:  PR[91,1] = PR[90,1] + 68.002;
   1:  PR[91,2] = PR[90,2] + -0.831;
   1:  PR[91,3] = PR[90,3] + 110.064;
   1:L PR[91] R[100]mm/sec CNT100;
   1:  PR[91,1] = PR[90,1] + 68.025;
   1:  PR[91,2] = PR[90,2] + -0.670;
   1:  PR[91,3] = PR[90,3] + 110.086;
   1:L PR[91] R[100]mm/sec CNT100;
   1:  PR[91,1] = PR[90,1] + 67.675;
   1:  PR[91,2] = PR[90,2] + 3.605;
   1:  PR[91,3] = PR[90,3] + 110.087;
   1:L PR[91] R[100]mm/sec CNT100;
   1:  PR[91,1] = PR[90,1] + 67.657;
   1:  PR[91,2] = PR[90,2] + 3.733;
   1:  PR[91,3] = PR[90,3] + 110.109;
   1:L PR[91] R[100]mm/sec CNT100;
   1:  PR[91,1] = PR[90,1] + 66.603;
   1:  PR[91,2] = PR[90,2] + 7.971;
   1:L PR[91] R[100]mm/sec CNT100;
   1:  PR[91,1] = PR[90,1] + 64.818;
   1:  PR[91,2] = PR[90,2] + 12.179;
   1:  PR[91,3] = PR[90,3] + 110.131;
   1:L PR[91] R[100]mm/sec CNT100;
   1:  PR[91,1] = PR[90,1] + 62.372;
   1:  PR[91,2] = PR[90,2] + 16.108;
   1:  PR[91,3] = PR[90,3] + 110.154;
   1:L PR[91] R[100]mm/sec CNT100;
   1:  PR[91,1] = PR[90,1] + 61.513;
   1:  PR[91,2] = PR[90,2] + 17.120;
   1:  PR[91,3] = PR[90,3] + 110.178;
   1:L PR[91] R[100]mm/sec CNT100;
   1:  PR[91,1] = PR[90,1] + 59.270;
   1:  PR[91,2] = PR[90,2] + 19.627;
   1:  PR[91,3] = PR[90,3] + 110.184;
   1:L PR[91] R[100]mm/sec CNT100;
   1:  PR[91,1] = PR[90,1] + 58.191;
   1:  PR[91,2] = PR[90,2] + 20.876;
   1:  PR[91,3] = PR[90,3] + 110.201;
   1:L PR[91] R[100]mm/sec CNT100;
   1:  PR[91,1] = PR[90,1] + 55.544;
   1:  PR[91,2] = PR[90,2] + 22.986;
   1:  PR[91,3] = PR[90,3] + 110.210;
   1:L PR[91] R[100]mm/sec CNT100;
   1:  PR[91,1] = PR[90,1] + 53.203;
   1:  PR[91,2] = PR[90,2] + 24.896;
   1:  PR[91,3] = PR[90,3] + 110.227;
   1:L PR[91] R[100]mm/sec CNT100;
   1:  PR[91,1] = PR[90,1] + 47.567;
   1:  PR[91,2] = PR[90,2] + 28.027;
   1:  PR[91,3] = PR[90,3] + 110.242;
   1:L PR[91] R[100]mm/sec CNT100;
   1:  PR[91,1] = PR[90,1] + 47.560;
   1:  PR[91,2] = PR[90,2] + 28.030;
   1:  PR[91,3] = PR[90,3] + 110.274;
   1:L PR[91] R[100]mm/sec CNT100;
   1:  PR[91,1] = PR[90,1] + 42.554;
   1:  PR[91,2] = PR[90,2] + 29.826;
   1:L PR[91] R[100]mm/sec CNT100;
   1:  PR[91,1] = PR[90,1] + 41.023;
   1:  PR[91,2] = PR[90,2] + 30.241;
   1:  PR[91,3] = PR[90,3] + 110.301;
   1:L PR[91] R[100]mm/sec CNT100;
   1:  PR[91,1] = PR[90,1] + 37.378;
   1:  PR[91,2] = PR[90,2] + 30.856;
   1:  PR[91,3] = PR[90,3] + 110.309;
   1:L PR[91] R[100]mm/sec CNT100;
   1:  PR[91,1] = PR[90,1] + 34.625;
   1:  PR[91,2] = PR[90,2] + 31.128;
   1:  PR[91,3] = PR[90,3] + 110.328;
   1:L PR[91] R[100]mm/sec CNT100;
   1:  PR[91,1] = PR[90,1] + 32.165;
   1:  PR[91,2] = PR[90,2] + 31.111;
   1:  PR[91,3] = PR[90,3] + 110.342;
   1:L PR[91] R[100]mm/sec CNT100;
   1:  PR[91,1] = PR[90,1] + 21.135;
   1:  PR[91,2] = PR[90,2] + 30.375;
   1:  PR[91,3] = PR[90,3] + 110.354;
   1:L PR[91] R[100]mm/sec CNT100;
   1:  PR[91,1] = PR[90,1] + 12.092;
   1:  PR[91,2] = PR[90,2] + 28.665;
   1:  PR[91,3] = PR[90,3] + 110.410;
   1:L PR[91] R[100]mm/sec CNT100;
   1:  PR[91,1] = PR[90,1] + 11.413;
   1:  PR[91,2] = PR[90,2] + 28.444;
   1:  PR[91,3] = PR[90,3] + 110.456;
   1:L PR[91] R[100]mm/sec CNT100;
   1:  PR[91,1] = PR[90,1] + 4.858;
   1:  PR[91,2] = PR[90,2] + 26.748;
   1:  PR[91,3] = PR[90,3] + 110.459;
   1:L PR[91] R[100]mm/sec CNT100;
   1:  PR[91,1] = PR[90,1] + -0.438;
   1:  PR[91,2] = PR[90,2] + 25.052;
   1:  PR[91,3] = PR[90,3] + 110.494;
   1:L PR[91] R[100]mm/sec CNT100;
   1:  PR[91,1] = PR[90,1] + -8.731;
   1:  PR[91,2] = PR[90,2] + 22.063;
   1:  PR[91,3] = PR[90,3] + 110.521;
   1:L PR[91] R[100]mm/sec CNT100;
   1:  PR[91,1] = PR[90,1] + -15.798;
   1:  PR[91,2] = PR[90,2] + 18.690;
   1:  PR[91,3] = PR[90,3] + 110.566;
   1:L PR[91] R[100]mm/sec CNT100;
   1:  PR[91,1] = PR[90,1] + -21.590;
   1:  PR[91,2] = PR[90,2] + 15.011;
   1:  PR[91,3] = PR[90,3] + 110.605;
   1:L PR[91] R[100]mm/sec CNT100;
   1:  PR[91,1] = PR[90,1] + -26.072;
   1:  PR[91,2] = PR[90,2] + 11.127;
   1:  PR[91,3] = PR[90,3] + 110.640;
   1:L PR[91] R[100]mm/sec CNT100;
   1:  PR[91,1] = PR[90,1] + -28.046;
   1:  PR[91,2] = PR[90,2] + 8.636;
   1:  PR[91,3] = PR[90,3] + 110.670;
   1:L PR[91] R[100]mm/sec CNT100;
   1:  PR[91,1] = PR[90,1] + -29.203;
   1:  PR[91,2] = PR[90,2] + 7.162;
   1:  PR[91,3] = PR[90,3] + 110.686;
   1:L PR[91] R[100]mm/sec CNT100 TB   .50sec,CALL END_PUD;
   1:  DO[117:Laser Start]=OFF;
   1:  PR[92] = PR[91];
   1:  PR[92,3] = PR[92,3] + 50;
   1:J PR[92] 10% FINE;
   1:  WAIT   5.00(sec);
   1:  DO[119:Gas]=OFF;
   1:  CALL HOME_ALL;
/POS
/END
